(* CoDeSys 2.3 export: VARTYPE_EXTCANQUEUE.EXP *)

(* Data type *)
TYPE VARTYPE_EXTCANQUEUE
STRUCT
	dummy : UINT;
	length: UINT;
	cobId : DWORD;
	rxData: ARRAY [0..7] OF USINT;
END_STRUCT
END_TYPE
